ABB RAPID module: LOGGER.mod

MODULE LOGGER

!////////////////
!GLOBAL VARIABLES
!////////////////
!PC communication
VAR socketdev clientSocket;
VAR socketdev serverSocket;
PERS string ipController;
PERS num loggerPort:= 5001;

!Robot configuration
PERS tooldata currentTool;
PERS wobjdata currentWobj;
VAR speeddata currentSpeed;
VAR zonedata currentZone;

!//Logger sampling rate
PERS num loggerWaitTime:= 0.02;  !Recommended for real controller
!PERS num loggerWaitTime:= 0.1;    !Recommended for virtual controller

PROC ServerCreateAndConnect(string ip, num port)
	VAR string clientIP;

	SocketCreate serverSocket;
	SocketBind serverSocket, ip, port;
	SocketListen serverSocket;
	TPWrite "LOGGER: Logger waiting for incomming connections ...";
	WHILE SocketGetStatus(clientSocket) <> SOCKET_CONNECTED DO
		SocketAccept serverSocket,clientSocket \ClientAddress:=clientIP \Time:=WAIT_MAX;
		IF SocketGetStatus(clientSocket) <> SOCKET_CONNECTED THEN
			TPWrite "LOGGER: Problem serving an incomming connection.";
			TPWrite "LOGGER: Try reconnecting.";
		ENDIF
		 !Wait 0.5 seconds for the next reconnection
		 WaitTime 0.5;
	ENDWHILE
	TPWrite "LOGGER: Connected to IP " + clientIP;
ENDPROC

PROC main()
	VAR string data;
	VAR robtarget position;
	VAR jointtarget joints;
    VAR string sendString;
	VAR bool connected;

	VAR string date;
	VAR string time;
	VAR clock timer;

    VAR num SensorX:=1;
    VAR num SensorY:=2;
    VAR num SensorZ:=3;
    VAR num SensorWX:=4;
    VAR num SensorWY:=5;
    VAR num SensorWZ:=6;
    VAR num ForceX:=7;
    VAR num ForceY:=8;
    VAR num ForceZ:=9;
    VAR num ForceWX:=10;
    VAR num ForceWY:=11;
    VAR num ForceWZ:=12;

	!//Torque Sensor Definitions
    TestSignDefine SensorX, 201, ROB_1, 1, 0;
    TestSignDefine SensorY, 202, ROB_1, 1, 0;
    TestSignDefine SensorZ, 203, ROB_1, 1, 0;
    TestSignDefine SensorWX, 204, ROB_1, 1, 0;
    TestSignDefine SensorWY, 205, ROB_1, 1, 0;
    TestSignDefine SensorWZ, 206, ROB_1, 1, 0;
    TestSignDefine ForceX, 207, ROB_1, 1, 0;
    TestSignDefine ForceY, 208, ROB_1, 1, 0;
    TestSignDefine ForceZ, 209, ROB_1, 1, 0;
    TestSignDefine ForceWX, 210, ROB_1, 1, 0;
    TestSignDefine ForceWY, 211, ROB_1, 1, 0;
    TestSignDefine ForceWZ, 212, ROB_1, 1, 0;


	date:= CDate();
	time:= CTime();
    ClkStart timer;

	connected:=FALSE;
	ServerCreateAndConnect ipController,loggerPort;
	connected:=TRUE;
	WHILE TRUE DO

		!Cartesian Coordinates
		position := CRobT(\Tool:=currentTool \WObj:=currentWObj);
		data := "# 0 ";
		data := data + date + " " + time + " ";
		data := data + NumToStr(ClkRead(timer),2) + " ";
		data := data + NumToStr(position.trans.x,1) + " ";
		data := data + NumToStr(position.trans.y,1) + " ";
		data := data + NumToStr(position.trans.z,1) + " ";
		data := data + NumToStr(position.rot.q1,3) + " ";
		data := data + NumToStr(position.rot.q2,3) + " ";
		data := data + NumToStr(position.rot.q3,3) + " ";
		data := data + NumToStr(position.rot.q4,3); !End of string
		IF connected = TRUE THEN
			SocketSend clientSocket \Str:=data;
		ENDIF
		WaitTime loggerWaitTime;

		!Joint Coordinates
		joints := CJointT();
		data := "# 1 ";
		data := data + date + " " + time + " ";
		data := data + NumToStr(ClkRead(timer),2) + " ";
		data := data + NumToStr(joints.robax.rax_1,2) + " ";
		data := data + NumToStr(joints.robax.rax_2,2) + " ";
		data := data + NumToStr(joints.robax.rax_3,2) + " ";
		data := data + NumToStr(joints.robax.rax_4,2) + " ";
		data := data + NumToStr(joints.robax.rax_5,2) + " ";
		data := data + NumToStr(joints.robax.rax_6,2); !End of string
		IF connected = TRUE THEN
			SocketSend clientSocket \Str:=data;
		ENDIF

		!Force Torque
		data := "# 2 ";
		data := data + date + " " + time + " ";
		data := data + NumToStr(ClkRead(timer),2) + " ";
		data := data + NumToStr(TestSignRead(SensorX),2) + " ";
		data := data + NumToStr(TestSignRead(SensorY),2) + " ";
		data := data + NumToStr(TestSignRead(SensorZ),2) + " ";
		data := data + NumToStr(TestSignRead(SensorWX),2) + " ";
		data := data + NumToStr(TestSignRead(SensorWY),2) + " ";
		data := data + NumToStr(TestSignRead(SensorWZ),2); !End of string
		IF connected = TRUE THEN
			SocketSend clientSocket \Str:=data;
		ENDIF

		WaitTime loggerWaitTime;
	ENDWHILE
	ERROR
	IF ERRNO=ERR_SOCK_CLOSED THEN
		TPWrite "LOGGER: Client has closed connection.";
	ELSE
		TPWrite "LOGGER: Connection lost: Unknown problem.";
	ENDIF
	connected:=FALSE;
	!Closing the server
	SocketClose clientSocket;
	SocketClose serverSocket;
	!Reinitiate the server
	ServerCreateAndConnect ipController,loggerPort;
	connected:= TRUE;
	RETRY;
ENDPROC

ENDMODULE
